FUNCTION_BLOCK DisableAllComponentsVisitor IMPLEMENTS I_ComponentVisitor
VAR
	Enablable : I_Enablable;
	_Enabled  : BOOL;
END_VAR

METHOD Disable
VAR_INPUT
	Components : I_ComponentCollection;
END_VAR
_Enabled := FALSE;
Components.Accept(THIS^);
END_METHOD

{attribute 'monitoring' := 'call'}
PROPERTY Enabled : BOOL
GET
Enabled := _Enabled;
END_GET
END_PROPERTY

METHOD VisitComponent
VAR_INPUT
	Component : I_Component;
END_VAR
IF __QUERYINTERFACE(Component, Enablable) THEN
	Enablable.Disable();
	IF Enablable.Enabled THEN
		_Enabled := TRUE;
	END_IF
END_IF
END_METHOD

END_FUNCTION_BLOCK

(* stored: Version 1.1.0.1, ProductVersion 3.1.4026.18
   POU DisableAllComponentsVisitor: Id {ef764682-9bc8-4f54-b748-2052670f038c}, SpecialFunc None
   Method Disable: Id {03e020e0-e181-4942-acf8-c3db1eade5e8}
   Property Enabled: Id {15fda2d7-913e-4794-bd9c-8bc9b08635f9}
   Get Get: Id {dbf2afbe-3425-4b81-9465-1ab0a61054d2}
   Method VisitComponent: Id {3266137d-7ebe-439a-839f-6f100fb8006e} *)
